{attribute 'enable_dynamic_creation'}	
TYPE S7_VARIABLE :
STRUCT
	Address : PVOID;
	Write : BOOL;
END_STRUCT
END_TYPE

(* stored: Version 1.1.0.1
   DUT S7_VARIABLE: Id {88b89260-c2ac-49de-a80f-3fa91ba3c246} *)
